{attribute addProperty BoxType "EK1100-0000-0018"}
{attribute addProperty Id "Beckhoff_EJ3xxxEK1122Beckhoff_EJ3xxxEK1122_6922078E162A_0001_EJ3004_0000_0019EJ3004_8D19A6A542052.5A_0002_EJ3004_0000_0020EJ3004_2BD8977C42052.5A_0003_EJ3004_0000_0021EJ3004_2BD8977C42052.5A_0004_EJ3048_0000_0020EJ3048_8660401635244A_0005_EJ3058_0000_0020EJ3058_8660401635244A_0006_EJ3068_0000_0020EJ3068_8660401635244A_0007_EJ3068_0000_0021EJ3068_8660401635244A_0008_EJ3104_0000_0019EJ3104_83515A0D22428A_0009_EJ3104_0000_0020EJ3104_83515A0D22428A_0010_EJ3104_0000_0021EJ3104_83515A0D22428A_0011_EJ3108_0000_0017EJ3108_8660401635244A_0012_EJ3108_0000_0018EJ3108_91E9C02235244A_0013_EJ3108_0000_0019EJ3108_91E9C02235244A_0014_EJ3202_0000_0019EJ3202_5359D6C325832.25A_0015_EJ3202_0000_0020EJ3202_5359D6C325832.25A_0016_EJ3202_0000_0021EJ3202_5359D6C325832.25A_0017_EJ3214_0000_0016EJ3214_6BC1D0AA22428A_0018_EJ3255_0000_0023EJ3255_A08AFE1A25632A_0019_EJ3318_0000_0017EJ3318_513179EA41652"}
{attribute addProperty CRC "2465498023"}
{attribute addProperty SizeInBites "6082"}
{attribute addProperty SizeInBytes "760.25"}
TYPE Beckhoff_EJ3xxx_92F483A7 EXTENDS EK1100_179A0949 :
STRUCT
	{attribute addProperty Name "Beckhoff_EJ3xxxEK1122"}
	Beckhoff_EJ3xxxEK1122 : Beckhoff_EJ3xxxEK1122_6922078E;
	{attribute addProperty Name "A_0001_EJ3004_0000_0019"}
	A_0001_EJ3004_0000_0019 : EJ3004_8D19A6A5;
	{attribute addProperty Name "A_0002_EJ3004_0000_0020"}
	A_0002_EJ3004_0000_0020 : EJ3004_2BD8977C;
	{attribute addProperty Name "A_0003_EJ3004_0000_0021"}
	A_0003_EJ3004_0000_0021 : EJ3004_2BD8977C;
	{attribute addProperty Name "A_0004_EJ3048_0000_0020"}
	A_0004_EJ3048_0000_0020 : EJ3048_86604016;
	{attribute addProperty Name "A_0005_EJ3058_0000_0020"}
	A_0005_EJ3058_0000_0020 : EJ3058_86604016;
	{attribute addProperty Name "A_0006_EJ3068_0000_0020"}
	A_0006_EJ3068_0000_0020 : EJ3068_86604016;
	{attribute addProperty Name "A_0007_EJ3068_0000_0021"}
	A_0007_EJ3068_0000_0021 : EJ3068_86604016;
	{attribute addProperty Name "A_0008_EJ3104_0000_0019"}
	A_0008_EJ3104_0000_0019 : EJ3104_83515A0D;
	{attribute addProperty Name "A_0009_EJ3104_0000_0020"}
	A_0009_EJ3104_0000_0020 : EJ3104_83515A0D;
	{attribute addProperty Name "A_0010_EJ3104_0000_0021"}
	A_0010_EJ3104_0000_0021 : EJ3104_83515A0D;
	{attribute addProperty Name "A_0011_EJ3108_0000_0017"}
	A_0011_EJ3108_0000_0017 : EJ3108_86604016;
	{attribute addProperty Name "A_0012_EJ3108_0000_0018"}
	A_0012_EJ3108_0000_0018 : EJ3108_91E9C022;
	{attribute addProperty Name "A_0013_EJ3108_0000_0019"}
	A_0013_EJ3108_0000_0019 : EJ3108_91E9C022;
	{attribute addProperty Name "A_0014_EJ3202_0000_0019"}
	A_0014_EJ3202_0000_0019 : EJ3202_5359D6C3;
	{attribute addProperty Name "A_0015_EJ3202_0000_0020"}
	A_0015_EJ3202_0000_0020 : EJ3202_5359D6C3;
	{attribute addProperty Name "A_0016_EJ3202_0000_0021"}
	A_0016_EJ3202_0000_0021 : EJ3202_5359D6C3;
	{attribute addProperty Name "A_0017_EJ3214_0000_0016"}
	A_0017_EJ3214_0000_0016 : EJ3214_6BC1D0AA;
	{attribute addProperty Name "A_0018_EJ3255_0000_0023"}
	A_0018_EJ3255_0000_0023 : EJ3255_A08AFE1A;
	{attribute addProperty Name "A_0019_EJ3318_0000_0017"}
	A_0019_EJ3318_0000_0017 : EJ3318_513179EA;
END_STRUCT
END_TYPE

(* stored: Version 1.2.0.0, ProductVersion 3.1.4024.9
   DUT Beckhoff_EJ3xxx_92F483A7: Id {c72a9466-63be-4af8-a811-73931b903471} *)
